PROGRAM MAIN
VAR
	bHalfSecondPulse													: BOOL;
	tonHalfSecPulse														: TON;
END_VAR

// Theseus - Main
// Rev 1.0 - September 31, 2024

P_M01.plc_version														:= '24_12_03_00';

/// TIMER PULSE
IF tonHalfSecPulse.Q THEN
	bHalfSecondPulse													:= NOT bHalfSecondPulse;
	tonHalfSecPulse(IN:= FALSE);
END_IF
tonHalfSecPulse(IN:= TRUE, PT:= T#500MS);

P_U01();
P_M01();
P_Alarms();

END_PROGRAM

(* stored: Version 1.1.0.1, ProductVersion 3.1.4024.12
   POU MAIN: Id {8c00b01f-f53f-430a-a974-d67c74f40a4b}, SpecialFunc None *)
